// Mitsubishi GX Works2 project: servo0914   PLC: Q03UDV

PROGRAM MAIN1
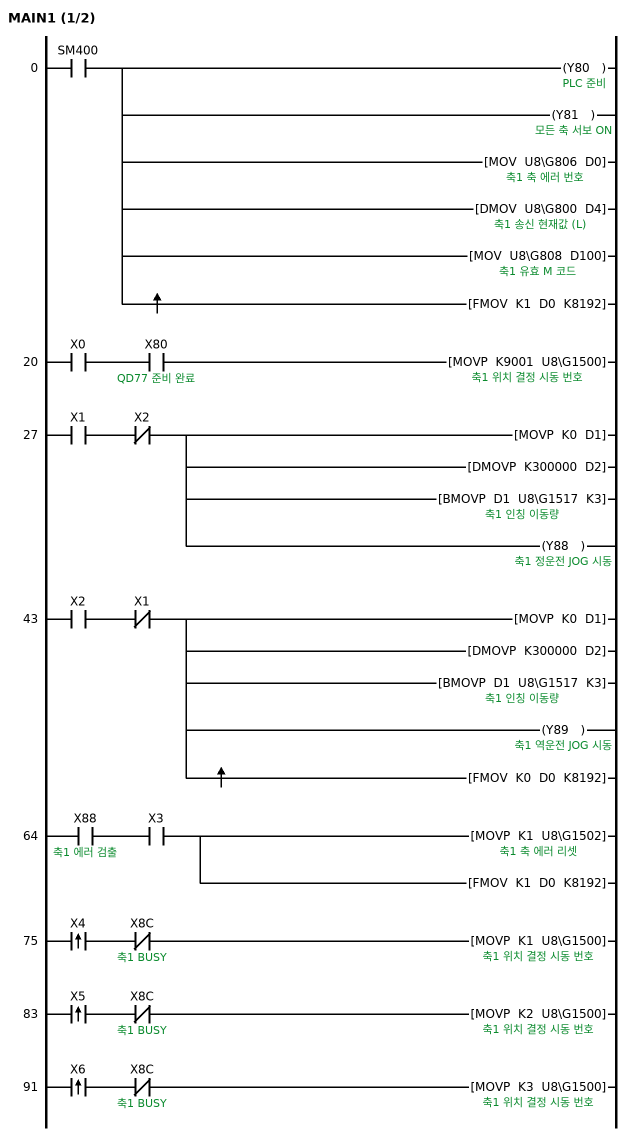
0     LD      SM400
      OUT     Y80  ; PLC 준비
      OUT     Y81  ; 모든 축 서보 ON
      MOV     U8\G806 D0  ; 축1 축 에러 번호
      DMOV    U8\G800 D4  ; 축1 송신 현재값 (L)
      MOV     U8\G808 D100  ; 축1 유효 M 코드
      MEP
      FMOV    K1 D0 K8192
20    LD      X0
      AND     X80  ; QD77 준비 완료
      MOVP    K9001 U8\G1500  ; 축1 위치 결정 시동 번호
27    LD      X1
      ANI     X2
      MOVP    K0 D1
      DMOVP   K300000 D2
      BMOVP   D1 U8\G1517 K3  ; 축1 인칭 이동량
      OUT     Y88  ; 축1 정운전 JOG 시동
43    LD      X2
      ANI     X1
      MOVP    K0 D1
      DMOVP   K300000 D2
      BMOVP   D1 U8\G1517 K3
      OUT     Y89  ; 축1 역운전 JOG 시동
      MEP
      FMOV    K0 D0 K8192
64    LD      X88  ; 축1 에러 검출
      AND     X3
      MOVP    K1 U8\G1502  ; 축1 축 에러 리셋
      FMOV    K1 D0 K8192
75    LDP     X4
      ANI     X8C  ; 축1 BUSY
      MOVP    K1 U8\G1500
83    LDP     X5
      ANI     X8C  ; 축1 BUSY
      MOVP    K2 U8\G1500
91    LDP     X6
      ANI     X8C  ; 축1 BUSY
      MOVP    K3 U8\G1500
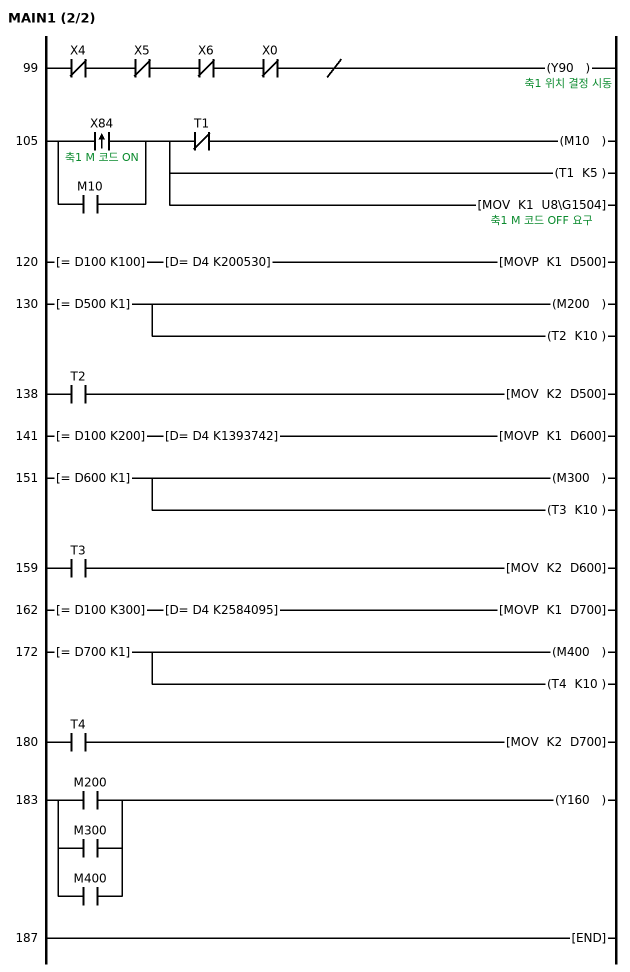
99    LDI     X4
      ANI     X5
      ANI     X6
      ANI     X0
      INV
      OUT     Y90  ; 축1 위치 결정 시동
105   LDP     X84  ; 축1 M 코드 ON
      OR      M10
      MPS
      ANI     T1
      OUT     M10
      MPP
      OUT     T1 K5
      MOV     K1 U8\G1504  ; 축1 M 코드 OFF 요구
120   LD=     D100 K100
      ANDD=   D4 K200530
      MOVP    K1 D500
130   LD=     D500 K1
      OUT     M200
      OUT     T2 K10
138   LD      T2
      MOV     K2 D500
141   LD=     D100 K200
      ANDD=   D4 K1393742
      MOVP    K1 D600
151   LD=     D600 K1
      OUT     M300
      OUT     T3 K10
159   LD      T3
      MOV     K2 D600
162   LD=     D100 K300
      ANDD=   D4 K2584095
      MOVP    K1 D700
172   LD=     D700 K1
      OUT     M400
      OUT     T4 K10
180   LD      T4
      MOV     K2 D700
183   LD      M200
      OR      M300
      OR      M400
      OUT     Y160
187   END
END_PROGRAM

// device comments not shown above
X81  ; 동기용 플래그
X85  ; 축2 M 코드 ON
X89  ; 축2 에러 검출
X8D  ; 축2 BUSY
X90  ; 축1 시동 완료
X91  ; 축2 시동 완료
X94  ; 축1 위치 결정 완료
X95  ; 축2 위치 결정 완료
Y84  ; 축1 축 정지
Y85  ; 축2 축 정지
Y8A  ; 축2 정운전 JOG 시동
Y8B  ; 축2 역운전 JOG 시동
Y91  ; 축2 위치 결정 시동
Y94  ; 축1 실행 금지 플래그
Y95  ; 축2 실행 금지 플래그
